TYPE DUT_RECIPE_USERPARAMETERINPUT :
STRUCT
	Value: REAL;
END_STRUCT
END_TYPE

(* stored: Version 1.1.0.1, ProductVersion 3.1.0.25
   DUT DUT_RECIPE_USERPARAMETERINPUT: Id {106cbfc7-f514-476b-be23-3eb28c1078b5} *)
